# EPICS substitutions: nasaAcqApp/Db/quartzAcq.substitutions
file "feed_base.template" {
{PREF="\$(P)GLD:", NAME="\$(P)GLD", ADDR="\$(IPADDR):803"}
}

file "goldenCtrl.template" {
{P="\$(P)"}
}

file "quartzAcqBase.template" {
{P="\$(P)", NAME="\$(NAME)", NELM="\$(NELM)"}
}

file "psc-psd.db" {
{N=01, P="\$(P)SA:Ch$(N):FFT:", NELM="\$(NELM)", INP="\$(P)SA:Ch$(N)_"}
{N=02, P="\$(P)SA:Ch$(N):FFT:", NELM="\$(NELM)", INP="\$(P)SA:Ch$(N)_"}
{N=03, P="\$(P)SA:Ch$(N):FFT:", NELM="\$(NELM)", INP="\$(P)SA:Ch$(N)_"}
{N=04, P="\$(P)SA:Ch$(N):FFT:", NELM="\$(NELM)", INP="\$(P)SA:Ch$(N)_"}
{N=05, P="\$(P)SA:Ch$(N):FFT:", NELM="\$(NELM)", INP="\$(P)SA:Ch$(N)_"}
{N=06, P="\$(P)SA:Ch$(N):FFT:", NELM="\$(NELM)", INP="\$(P)SA:Ch$(N)_"}
{N=07, P="\$(P)SA:Ch$(N):FFT:", NELM="\$(NELM)", INP="\$(P)SA:Ch$(N)_"}
{N=08, P="\$(P)SA:Ch$(N):FFT:", NELM="\$(NELM)", INP="\$(P)SA:Ch$(N)_"}
{N=09, P="\$(P)SA:Ch$(N):FFT:", NELM="\$(NELM)", INP="\$(P)SA:Ch$(N)_"}
{N=10, P="\$(P)SA:Ch$(N):FFT:", NELM="\$(NELM)", INP="\$(P)SA:Ch$(N)_"}
{N=11, P="\$(P)SA:Ch$(N):FFT:", NELM="\$(NELM)", INP="\$(P)SA:Ch$(N)_"}
{N=12, P="\$(P)SA:Ch$(N):FFT:", NELM="\$(NELM)", INP="\$(P)SA:Ch$(N)_"}
{N=13, P="\$(P)SA:Ch$(N):FFT:", NELM="\$(NELM)", INP="\$(P)SA:Ch$(N)_"}
{N=14, P="\$(P)SA:Ch$(N):FFT:", NELM="\$(NELM)", INP="\$(P)SA:Ch$(N)_"}
{N=15, P="\$(P)SA:Ch$(N):FFT:", NELM="\$(NELM)", INP="\$(P)SA:Ch$(N)_"}
{N=16, P="\$(P)SA:Ch$(N):FFT:", NELM="\$(NELM)", INP="\$(P)SA:Ch$(N)_"}
{N=17, P="\$(P)SA:Ch$(N):FFT:", NELM="\$(NELM)", INP="\$(P)SA:Ch$(N)_"}
{N=18, P="\$(P)SA:Ch$(N):FFT:", NELM="\$(NELM)", INP="\$(P)SA:Ch$(N)_"}
{N=19, P="\$(P)SA:Ch$(N):FFT:", NELM="\$(NELM)", INP="\$(P)SA:Ch$(N)_"}
{N=20, P="\$(P)SA:Ch$(N):FFT:", NELM="\$(NELM)", INP="\$(P)SA:Ch$(N)_"}
{N=21, P="\$(P)SA:Ch$(N):FFT:", NELM="\$(NELM)", INP="\$(P)SA:Ch$(N)_"}
{N=22, P="\$(P)SA:Ch$(N):FFT:", NELM="\$(NELM)", INP="\$(P)SA:Ch$(N)_"}
{N=23, P="\$(P)SA:Ch$(N):FFT:", NELM="\$(NELM)", INP="\$(P)SA:Ch$(N)_"}
{N=24, P="\$(P)SA:Ch$(N):FFT:", NELM="\$(NELM)", INP="\$(P)SA:Ch$(N)_"}
{N=25, P="\$(P)SA:Ch$(N):FFT:", NELM="\$(NELM)", INP="\$(P)SA:Ch$(N)_"}
{N=26, P="\$(P)SA:Ch$(N):FFT:", NELM="\$(NELM)", INP="\$(P)SA:Ch$(N)_"}
{N=27, P="\$(P)SA:Ch$(N):FFT:", NELM="\$(NELM)", INP="\$(P)SA:Ch$(N)_"}
{N=28, P="\$(P)SA:Ch$(N):FFT:", NELM="\$(NELM)", INP="\$(P)SA:Ch$(N)_"}
{N=29, P="\$(P)SA:Ch$(N):FFT:", NELM="\$(NELM)", INP="\$(P)SA:Ch$(N)_"}
{N=30, P="\$(P)SA:Ch$(N):FFT:", NELM="\$(NELM)", INP="\$(P)SA:Ch$(N)_"}
{N=31, P="\$(P)SA:Ch$(N):FFT:", NELM="\$(NELM)", INP="\$(P)SA:Ch$(N)_"}
{N=32, P="\$(P)SA:Ch$(N):FFT:", NELM="\$(NELM)", INP="\$(P)SA:Ch$(N)_"}
}

file "quartzAcqChan.template" {
{N=01,  OFF=40,  P="\$(P)", NAME="\$(NAME)", NELM="\$(NELM)", FLNK="$(P)SA:Ch02_"}
{N=02,  OFF=43,  P="\$(P)", NAME="\$(NAME)", NELM="\$(NELM)", FLNK="$(P)SA:Ch03_"}
{N=03,  OFF=46,  P="\$(P)", NAME="\$(NAME)", NELM="\$(NELM)", FLNK="$(P)SA:Ch04_"}
{N=04,  OFF=49,  P="\$(P)", NAME="\$(NAME)", NELM="\$(NELM)", FLNK="$(P)SA:Ch05_"}
{N=05,  OFF=52,  P="\$(P)", NAME="\$(NAME)", NELM="\$(NELM)", FLNK="$(P)SA:Ch06_"}
{N=06,  OFF=55,  P="\$(P)", NAME="\$(NAME)", NELM="\$(NELM)", FLNK="$(P)SA:Ch07_"}
{N=07,  OFF=58,  P="\$(P)", NAME="\$(NAME)", NELM="\$(NELM)", FLNK="$(P)SA:Ch08_"}
{N=08,  OFF=61,  P="\$(P)", NAME="\$(NAME)", NELM="\$(NELM)", FLNK="$(P)SA:Ch09_"}
{N=09,  OFF=64,  P="\$(P)", NAME="\$(NAME)", NELM="\$(NELM)", FLNK="$(P)SA:Ch10_"}
{N=10,  OFF=67,  P="\$(P)", NAME="\$(NAME)", NELM="\$(NELM)", FLNK="$(P)SA:Ch11_"}
{N=11,  OFF=70,  P="\$(P)", NAME="\$(NAME)", NELM="\$(NELM)", FLNK="$(P)SA:Ch12_"}
{N=12,  OFF=73,  P="\$(P)", NAME="\$(NAME)", NELM="\$(NELM)", FLNK="$(P)SA:Ch13_"}
{N=13,  OFF=76,  P="\$(P)", NAME="\$(NAME)", NELM="\$(NELM)", FLNK="$(P)SA:Ch14_"}
{N=14,  OFF=79,  P="\$(P)", NAME="\$(NAME)", NELM="\$(NELM)", FLNK="$(P)SA:Ch15_"}
{N=15,  OFF=82,  P="\$(P)", NAME="\$(NAME)", NELM="\$(NELM)", FLNK="$(P)SA:Ch16_"}
{N=16,  OFF=85,  P="\$(P)", NAME="\$(NAME)", NELM="\$(NELM)", FLNK="$(P)SA:Ch17_"}
{N=17,  OFF=88,  P="\$(P)", NAME="\$(NAME)", NELM="\$(NELM)", FLNK="$(P)SA:Ch18_"}
{N=18,  OFF=91,  P="\$(P)", NAME="\$(NAME)", NELM="\$(NELM)", FLNK="$(P)SA:Ch19_"}
{N=19,  OFF=94,  P="\$(P)", NAME="\$(NAME)", NELM="\$(NELM)", FLNK="$(P)SA:Ch20_"}
{N=20,  OFF=97,  P="\$(P)", NAME="\$(NAME)", NELM="\$(NELM)", FLNK="$(P)SA:Ch21_"}
{N=21,  OFF=100,  P="\$(P)", NAME="\$(NAME)", NELM="\$(NELM)", FLNK="$(P)SA:Ch22_"}
{N=22,  OFF=103,  P="\$(P)", NAME="\$(NAME)", NELM="\$(NELM)", FLNK="$(P)SA:Ch23_"}
{N=23,  OFF=106,  P="\$(P)", NAME="\$(NAME)", NELM="\$(NELM)", FLNK="$(P)SA:Ch24_"}
{N=24,  OFF=109,  P="\$(P)", NAME="\$(NAME)", NELM="\$(NELM)", FLNK="$(P)SA:Ch25_"}
{N=25,  OFF=112,  P="\$(P)", NAME="\$(NAME)", NELM="\$(NELM)", FLNK="$(P)SA:Ch26_"}
{N=26,  OFF=115,  P="\$(P)", NAME="\$(NAME)", NELM="\$(NELM)", FLNK="$(P)SA:Ch27_"}
{N=27,  OFF=118,  P="\$(P)", NAME="\$(NAME)", NELM="\$(NELM)", FLNK="$(P)SA:Ch28_"}
{N=28,  OFF=121,  P="\$(P)", NAME="\$(NAME)", NELM="\$(NELM)", FLNK="$(P)SA:Ch29_"}
{N=29,  OFF=124,  P="\$(P)", NAME="\$(NAME)", NELM="\$(NELM)", FLNK="$(P)SA:Ch30_"}
{N=30,  OFF=127,  P="\$(P)", NAME="\$(NAME)", NELM="\$(NELM)", FLNK="$(P)SA:Ch31_"}
{N=31,  OFF=130,  P="\$(P)", NAME="\$(NAME)", NELM="\$(NELM)", FLNK="$(P)SA:Ch32_"}
{N=32,  OFF=133,  P="\$(P)", NAME="\$(NAME)", NELM="\$(NELM)", FLNK="$(P)SA:HldOff_"}
}
